(* PLC project Unnamed, Unknown Unnamed 1 *)
(* stored: creationDateTime 2025-11-02T14:36:43, modificationDateTime 2025-11-02T14:49:10 *)

TYPE MotorControlType : STRUCT
  MotorOn : BOOL := False;
END_STRUCT;
END_TYPE

PROGRAM MotorControl
  VAR
    I_StartPB : BOOL := False;
    I_StopPB : BOOL := False;
    F_MotorStarted : BOOL := False;
    F_MotorStopped : BOOL := False;
  END_VAR
  VAR_EXTERNAL
    MotorControlGlobal : MotorControlType;
  END_VAR

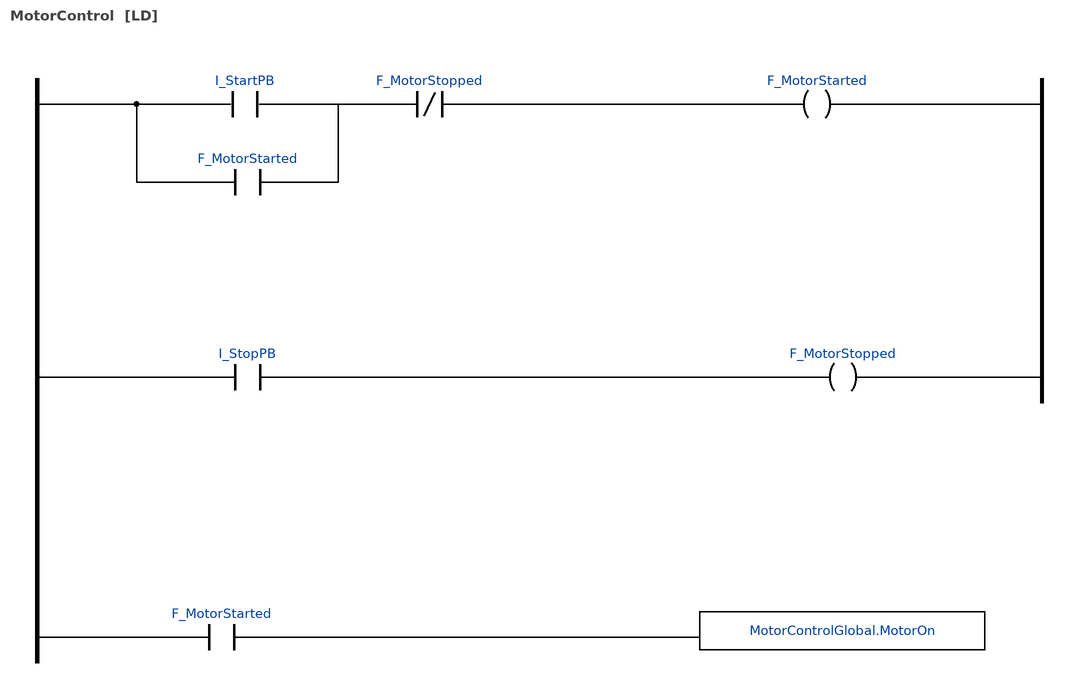
(* LD diagram, written out as Structured Text *)
F_MotorStarted := (I_StartPB OR F_MotorStarted) AND NOT F_MotorStopped;
F_MotorStopped := I_StopPB;
MotorControlGlobal.MotorOn := F_MotorStarted;
END_PROGRAM

PROGRAM Outputs
  VAR_OUTPUT
    Q_Motor : BOOL;
  END_VAR
  VAR_EXTERNAL
    MotorControlGlobal : MotorControlType;
  END_VAR

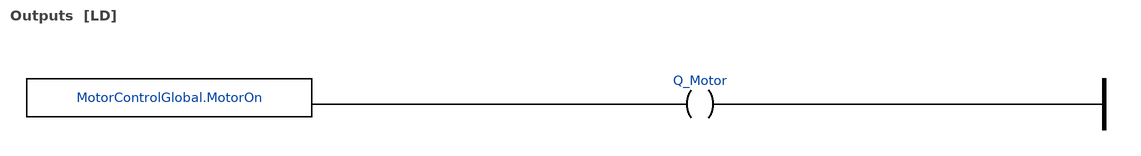
(* LD diagram, written out as Structured Text *)
Q_Motor := MotorControlGlobal.MotorOn;
END_PROGRAM

CONFIGURATION Config0
  VAR_GLOBAL
    MotorControlGlobal : MotorControlType;
  END_VAR
  RESOURCE Res0 ON PLC
    TASK task0(INTERVAL := T#20ms, PRIORITY := 0);
    PROGRAM MotorControlInstance WITH task0 : MotorControl;
    PROGRAM OutPutInstance WITH task0 : Outputs;
  END_RESOURCE
END_CONFIGURATION
